Universal Robots PolyScope program: g_full_bow.urp

Program g_full_bow (installation=string_planes directory=/programs/strings createdIn=5.17.3 lastSavedIn=5.17.3 robotSerialNumber=20245501435)
Calibrated DH parameters: a=[0.000154, -0.137004, -0.385524, -0.00002, 0.000092, 0]; d=[0.162441, 211.794786, -230.585024, 18.923638, 0.099786, 0.09951]; alpha=[1.569493, -0.001902, 0.003874, 1.570111, -1.570167, 0]; deltaTheta=[0, -1.242934, 1.056292, 0.186646, 0.000002, 0.000001]
InitVariablesNode
Robot Program (runOnlyOnce=false)
  MoveL speed 250 mm/s, acceleration 1200 mm/s^2 (useActiveTCP=true) feature=Base
    Waypoint Waypoint_1: TCP in base x=295.799 y=651.768 z=117.422 mm, rx=-1.6921 ry=-1.7553 rz=0.606 rad; joints [-130.58, -31.353, 78.738, -108.525, -53.252, -142.213] deg; TCP offset x=28.21 y=-96.107 z=-99.69 mm, rx=0 ry=0 rz=0 rad
    Waypoint Waypoint_2: TCP in base x=242.21 y=182.121 z=104.888 mm, rx=-1.6706 ry=-1.8173 rz=0.7575 rad; joints [-175.135, -52.326, 143.099, -134.271, -88.413, -180.293] deg
  MoveL speed 250 mm/s, acceleration 1200 mm/s^2 (useActiveTCP=true) feature=Base
    Waypoint Waypoint_2: TCP in base x=242.21 y=182.121 z=104.888 mm, rx=-1.6706 ry=-1.8173 rz=0.7575 rad; joints [-175.135, -52.326, 143.099, -134.271, -88.413, -180.293] deg
    Waypoint Waypoint_1: TCP in base x=295.799 y=651.768 z=117.422 mm, rx=-1.6921 ry=-1.7553 rz=0.606 rad; joints [-130.58, -31.353, 78.738, -108.525, -53.252, -142.213] deg
  Wait Sleep waitTime=300
  bow_dir := True
  note_dur := 1
  Timer (action=Start) variable(name=timer_1)
  If bow_dir
    MoveL speed 250 mm/s, acceleration 1200 mm/s^2 (useActiveTCP=true) feature=Base
      Waypoint Waypoint_2: TCP in base x=242.21 y=182.121 z=104.888 mm, rx=-1.6706 ry=-1.8173 rz=0.7575 rad; joints [-175.135, -52.326, 143.099, -134.271, -88.413, -180.293] deg
        Until EXPRESSION (allowActions=false) ExpressionBranch=timer_1≟note_dur
  Else 
    MoveL speed 250 mm/s, acceleration 1200 mm/s^2 (useActiveTCP=true) feature=Base
      Waypoint Waypoint_1: TCP in base x=295.799 y=651.768 z=117.422 mm, rx=-1.6921 ry=-1.7553 rz=0.606 rad; joints [-130.58, -31.353, 78.738, -108.525, -53.252, -142.213] deg
        Until EXPRESSION (allowActions=false) ExpressionBranch=timer_1≟note_dur
  SuppressedNode
    MoveL speed 250 mm/s, acceleration 1200 mm/s^2 (useActiveTCP=true) feature=Base
      Waypoint Waypoint_1: TCP in base x=333.313 y=655.49 z=103.651 mm, rx=-1.6491 ry=-1.7982 rz=0.6657 rad; joints [-132.463, -27.757, 71.844, -100.482, -56.044, -147.729] deg
      Waypoint Waypoint_3: motionParameters(blendRadius=0.05); TCP in base x=267.763 y=455.808 z=63.345 mm, rx=-1.6064 ry=-1.9107 rz=0.8702 rad; joints [-141.616, -39.193, 108.914, -115.288, -70.782, -159.12] deg
      Waypoint Waypoint_2: TCP in base x=243.61 y=214.062 z=64.413 mm, rx=-1.5874 ry=-1.9212 rz=0.9621 rad; joints [-169.308, -44.602, 138.126, -133.88, -94.42, -177.775] deg
  Timer (action=Stop) variable=timer_1
  Timer (action=Reset) variable=timer_1
